// Mitsubishi GX Works2 project: TIMMER1   PLC: Q03UDV

PROGRAM MAIN
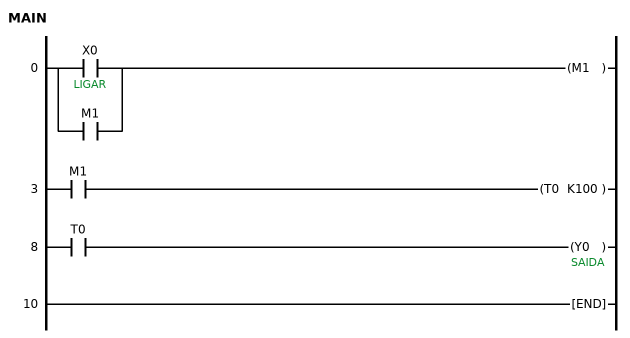
0     LD      X0  ; LIGAR
      OR      M1
      OUT     M1
3     LD      M1
      OUT     T0 K100
8     LD      T0
      OUT     Y0  ; SAIDA
10    END
END_PROGRAM

// device comments not shown above
X1  ; DESLIGAR
